INTERFACE INTERNAL I_DomainInternal EXTENDS I_Domain

PROPERTY CTable : I_CTable
GET
END_GET
END_PROPERTY

PROPERTY INTERNAL IsRegistered : BOOL
GET
END_GET
SET
END_SET
END_PROPERTY

END_INTERFACE

(* stored: Version 1.1.0.1
   Itf I_DomainInternal: Id {6083b3e1-a52a-4adb-ab93-b067bb8e3843}
   Property CTable: Id {dec401c4-4383-4519-9989-360a8fdd0d50}
   Get Get: Id {e638ad6f-302d-411a-b3f5-c62c71136055}
   Property IsRegistered: Id {bd0895a8-f3a0-4b4a-ae25-8af0498bbcad}
   Get Get: Id {4675dedf-552d-4053-93cc-82e6cd1dc776}
   Set Set: Id {da956018-1dba-4d32-b88c-848e5ba18d5f} *)
